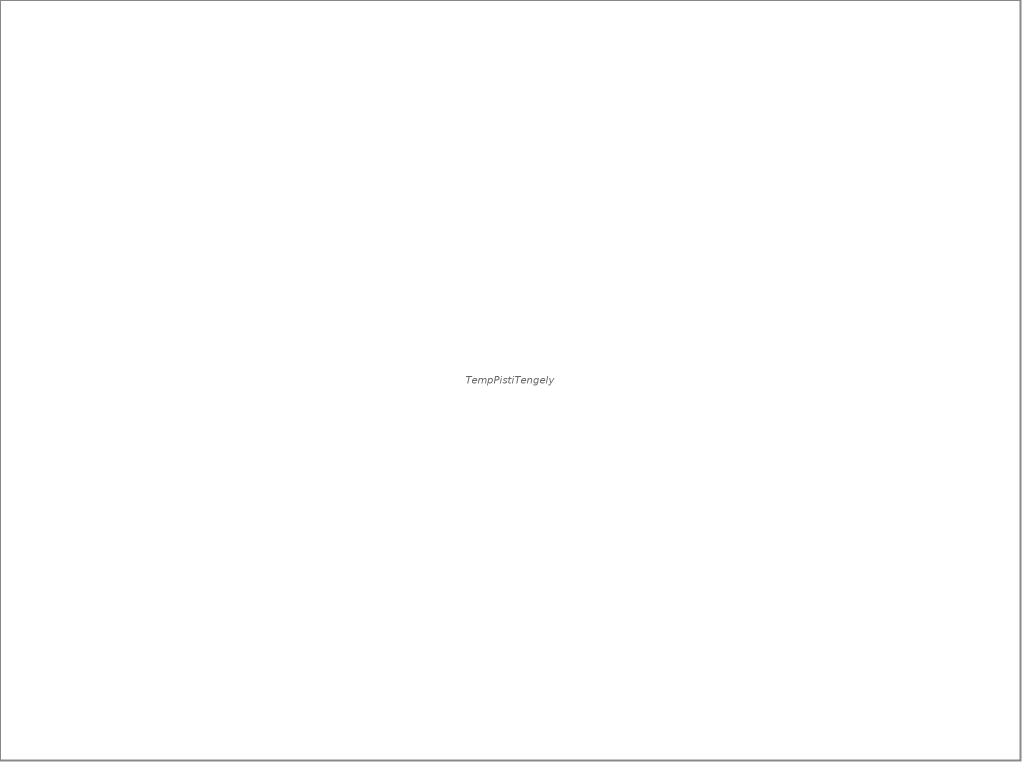
VISUALIZATION TempPisti  // 1022x762
    TabControl (0,0 1020x760)
        shows TempPistiTengely()
        shows TempPistiBehelyezes()
        shows TempPistiHegesztes()
        shows TempPistiKappe()
        shows TempPistiVegmero()
        shows Kodolvaso()
        [0]: TabTitle=Tengely
        [1]: TabTitle=Behelyezés
        [2]: TabTitle=Hegesztés
        [3]: TabTitle=Kappézás
        [4]: TabTitle=Végmérő
        [5]: TabTitle=Kódolvasó
END_VISUALIZATION

(* stored: Version 1.1.0.1, ProductVersion 3.1.4024.11
   Visu TempPisti: Id {81094e82-2082-420e-b74f-53f3c0c34354} *)
